// SIMATIC S7-200 project (STEP 7-Micro/WIN), CPU 226 REL 01.00

SYMBOL_TABLE SYM1
就联开关_就地甲I00      I0.0
就联开关_就地乙I01      I0.1
碎煤一开关_正转I02      I0.2
碎煤一开关_反转I03      I0.3
采样头开关_接通I04      I0.4
给料缩分机开关_接通I05    I0.5
提升螺旋机开关_接通I06    I0.6
联动信号甲I07         I0.7
联动信号乙I10         I1.0
采样甲限位I11         I1.1
采样乙限位I12         I1.2
分样机检测I13         I1.3
提升机热继I14         I1.4
螺旋机热继I15         I1.5
碎煤机一热继I16        I1.6
液压颚热继I17         I1.7
给料缩分机热继I20       I2.0
采样头甲热继I21        I2.1
采样头乙热继I22        I2.2
碎煤机二热继I23        I2.3
二级螺旋热继I24        I2.4
分样盘热继I25         I2.5
碎煤机一过流I26        I2.6
启动输入I27          I2.7
碎煤二开关_正转I30      I3.0
碎煤二开关_反转I31      I3.1
分样按钮_接通I32       I3.2
碎煤机二过流I33        I3.3
提升机_输出Q00        Q0.0
螺旋机_输出Q01        Q0.1
碎煤一正_输出QO2       Q0.2
碎煤一反_输出Q03       Q0.3
液压颚_输出Q04        Q0.4
给料机_输出Q05        Q0.5
采样甲_输出Q06        Q0.6
采样乙_输出Q07        Q0.7
缩分器_输出Q10        Q1.0
系统启动Q11          Q1.1
输煤带甲指示Q12        Q1.2
报警指示Q13          Q1.3
输煤带乙指示Q14        Q1.4
碎煤二正_输出Q16       Q1.6
碎煤二反_输出Q17       Q1.7
二级螺旋正_输出Q20      Q2.0
二级螺旋反_输出Q21      Q2.1
分样机_输出Q22        Q2.2
END_SYMBOL_TABLE

ORGANIZATION_BLOCK MAIN:OB1
TITLE=系统部署在洛河某燃煤处理车间。
// 采样过程从煤炭提升开始，提升机将煤炭送至高处，但只有在提升机热继未动作时才会启动，以保护设备。提升机在系统投运时，根据提升螺旋机开关_接通的状态启动，并通过运行指示显示其工作状态。随后，螺旋机在系统投运一段时间后（由计时触发），根据提升螺旋机开关_接通的状态并确保螺旋机热继正常，将煤炭输送至破碎区。螺旋机的运行状态通过显示实时反馈给操作员，确保输送过程可监控。
// 煤炭进入破碎环节，碎煤一正和碎煤二正依次破碎大块煤炭。若碎煤机一过流检测到堵塞，系统自动切换至碎煤一反反转排除故障，反转仅在过流或手动触发时发生，确保系统连续运行。碎煤一正的正转状态通过显示反馈，方便操作员确认破碎进程。破碎过程中，液压颚在碎煤一正运行时周期性动作，控制煤炭流量，其运行时间由液压间隔时间和击时间精确调节，避免设备过载。破碎后的煤炭通过给料机调节流量，进入采样区。
// 采样环节由采样甲和采样乙执行，根据采样间隔时间周期性采集样品，避免采样频率过高。采样甲完成标志在采样甲限位触发时记录，标记采样头甲的任务结束。采集的样品经缩分器处理后，由二级螺旋正输送，最终通过手动触发分样按钮_接通启动分样机。分样机在系统投运标志激活且采样完成后，根据分样按钮_接通的指令，将样品分配到不同容器中。分样机的运行状态通过显示提供给操作员，便于监控样品分配过程。每台设备的启动都依赖对应热继未动作，确保安全运行。若发生故障，如碎煤机一热继或碎煤机二过流，系统立即触发报警指示，报警状态持续显示，直到复位标志被触发以清除故障记录。复位标志在触发后清除故障记录，为系统恢复正常操作做准备，此时设备保持当前运行状态等待进一步操作。
// 
// 
BEGIN
Network 1 // 洛河入炉煤程序
// 段注释
// 
LD     SM5.0
STOP
Network 2
LD     SM0.1
LD     系统启动Q11:Q1.1
EU
OLD
R      M0.7, 1
R      M1.1, 1
R      M1.2, 1
R      M5.1, 1
R      M5.4, 1
Network 3
LDN    提升机热继I14:I1.4
AN     螺旋机热继I15:I1.5
AN     碎煤机一热继I16:I1.6
AN     液压颚热继I17:I1.7
AN     给料缩分机热继I20:I2.0
AN     采样头甲热继I21:I2.1
AN     采样头乙热继I22:I2.2
AN     碎煤机二热继I23:I2.3
AN     二级螺旋热继I24:I2.4
AN     分样盘热继I25:I2.5
=      M0.1
Network 4
LD     启动输入I27:I2.7
A      M0.1
AN     M5.0
TON    T101, +2
Network 5
LD     T101
=      系统启动Q11:Q1.1
Network 6 // 显待机
// 
// 
LD     系统启动Q11:Q1.1
AN     M2.0
BMB    VB420, VB40, 20
Network 7 // 显示停止
// 
// 
LDN    系统启动Q11:Q1.1
BMB    VB520, VB40, 20
Network 8 // 系统投运
// 
// 
LD     就联开关_就地甲I00:I0.0
O      就联开关_就地乙I01:I0.1
LDN    就联开关_就地甲I00:I0.0
AN     就联开关_就地乙I01:I0.1
LD     联动信号甲I07:I0.7
O      联动信号乙I10:I1.0
ALD
OLD
O      M2.0
A      系统启动Q11:Q1.1
AN     M1.4
=      M2.0
BMB    VB400, VB40, 10
TON    T127, +10
TON    T128, +20
TON    T129, +50
EU
R      M20.2, 1
R      M20.3, 1
Network 9 // 显示甲侧
// 
// 
LD     就联开关_就地甲I00:I0.0
BMB    VB740, VB260, 10
Network 10 // 显示乙侧
// 
// 
LD     就联开关_就地乙I01:I0.1
BMB    VB760, VB260, 10
Network 11 // 显示联动
// 
// 
LDN    就联开关_就地甲I00:I0.0
AN     就联开关_就地乙I01:I0.1
BMB    VB780, VB260, 10
Network 12 // 分计时器
// 
// 
LD     M2.0
AN     T115
TON    T115, +600
MOVW   T115, VW340
/I     +10, VW340
Network 13 // 一小时定时器
// 
// 
LD     T115
LD     C1
O      SM0.1
CTU    C1, +60
Network 14
LD     M2.0
MOVW   C1, VW342
Network 15
LD     M2.0
EU
MOVW   VW344, VW344
MOVW   +0, VW312
MOVW   +0, VW314
Network 16 // 累计运行时间记录
// 
// 
LD     C1
EU
INCW   VW344
INCW   VW346
Network 17 // 设置停机延时时间
// 
// 
LD     SM0.0
MOVW   VW396, AC0
MUL    +10, AC0
MOVW   AC0, VW398
Network 18 // 停运指令后启动30秒延时
// 
// 
LD     系统启动Q11:Q1.1
A      M2.0
AN     就联开关_就地甲I00:I0.0
AN     就联开关_就地乙I01:I0.1
AN     联动信号甲I07:I0.7
AN     联动信号乙I10:I1.0
TON    T113, VW398
Network 19 // M1.4去停机,T105为反排结束;如果碎煤机不在"正转"位置,就不执行反排动作而直接停机.
// 
// 
LD     T113
LDN    碎煤一开关_正转I02:I0.2
O      T105
ALD
LDN    碎煤二开关_正转I30:I3.0
O      T123
ALD
EU
=      M1.4
Network 20 // 甲启动状态，
// 
// 
LD     就联开关_就地甲I00:I0.0
=      M20.0
Network 21 // 乙启动状态，送远方Q2。5
// 
// 
LD     就联开关_就地乙I01:I0.1
=      M20.1
Network 22 // 甲侧初始状态
// 
// 
LDN    就联开关_就地甲I00:I0.0
AN     就联开关_就地乙I01:I0.1
A      联动信号甲I07:I0.7
A      M2.0
EU
AN     M20.3
S      M20.2, 1
R      M20.3, 1
Network 23 // 乙侧初始状态
// 
// 
LDN    就联开关_就地甲I00:I0.0
AN     就联开关_就地乙I01:I0.1
A      联动信号乙I10:I1.0
A      M2.0
EU
AN     M20.2
S      M20.3, 1
R      M20.2, 1
Network 24 // 双皮带同时运行情况，从双皮带变为单皮带情况。
// 
// 
LDN    就联开关_就地甲I00:I0.0
AN     就联开关_就地乙I01:I0.1
LPS
A      联动信号甲I07:I0.7
A      联动信号乙I10:I1.0
LPS
AN     M20.2
TON    T131, +18000
LRD
AN     M20.3
TON    T132, +18000
LRD
A      T131
S      M20.2, 1
R      M20.3, 1
LPP
A      T132
S      M20.3, 1
R      M20.2, 1
LPP
LPS
A      联动信号甲I07:I0.7
ED
S      M20.3, 1
R      M20.2, 1
LPP
A      联动信号乙I10:I1.0
ED
S      M20.2, 1
R      M20.3, 1
Network 25 // 二级螺旋
// 
// 
LD     M20.1
O      M20.3
A      M2.0
A      提升螺旋机开关_接通I06:I0.6
AN     二级螺旋热继I24:I2.4
AN     二级螺旋正_输出Q20:Q2.0
=      二级螺旋反_输出Q21:Q2.1
Network 26 // 二级螺旋正转指示
// 
// 
LD     二级螺旋正_输出Q20:Q2.0
LPS
A      SM0.6
LPS
AW<=   VW392, +0
MOVW   +100, VW392
LPP
DECW   VW392
LPP
NOT
MOVW   +0, VW392
Network 27 // 二级螺旋反转指示
// 
// 
LD     二级螺旋反_输出Q21:Q2.1
LPS
A      SM0.6
LPS
AW<=   VW394, +0
MOVW   +100, VW394
LPP
DECW   VW394
LPP
NOT
MOVW   +0, VW394
Network 28
LD     二级螺旋正_输出Q20:Q2.0
BMB    VB440, VB60, 20
Network 29
LD     二级螺旋反_输出Q21:Q2.1
BMB    VB460, VB60, 20
Network 30
LDN    二级螺旋正_输出Q20:Q2.0
AN     二级螺旋反_输出Q21:Q2.1
BMB    VB480, VB60, 20
Network 31 // 提升机启动.
// 
// 
LD     M2.0
A      提升螺旋机开关_接通I06:I0.6
AN     提升机热继I14:I1.4
LPS
=      提升机_输出Q00:Q0.0
A      SM0.6
LPS
AW<=   VW390, +0
MOVW   +100, VW390
LPP
DECW   VW390
LPP
NOT
MOVW   +100, VW390
Network 32 // 提升机运行
// 
// 
LD     提升机_输出Q00:Q0.0
BMB    VB500, VB80, 20
Network 33 // 提升机停机
// 
// 
LDN    提升机_输出Q00:Q0.0
AN     提升机热继I14:I1.4
BMB    VB520, VB80, 20
Network 34 // 提升机故障
// 
// 
LD     提升机热继I14:I1.4
BMB    VB540, VB80, 20
Network 35 // 螺旋机一启动.
// 
// 
LD     T127
AN     螺旋机热继I15:I1.5
A      提升螺旋机开关_接通I06:I0.6
=      螺旋机_输出Q01:Q0.1
Network 36 // 螺旋一运行
// 
// 
LD     螺旋机_输出Q01:Q0.1
BMB    VB500, VB100, 20
Network 37 // 螺旋一停机
// 
// 
LDN    螺旋机_输出Q01:Q0.1
AN     螺旋机热继I15:I1.5
BMB    VB520, VB100, 20
Network 38 // 螺旋一故障
// 
// 
LD     螺旋机热继I15:I1.5
BMB    VB540, VB100, 20
Network 39 // 碎煤机
// 
// 
LD     T128
A      碎煤一开关_正转I02:I0.2
AN     碎煤机一热继I16:I1.6
AN     M0.5
TON    T102, +20
A      T102
LPS
=      碎煤一正_输出QO2:Q0.2
A      SM0.6
LPS
AW<=   VW378, +0
MOVW   +100, VW378
LPP
DECW   VW378
LPP
NOT
MOVW   +0, VW378
Network 40 // 碎煤机过流防扰
// 
// 
LD     M2.0
A      碎煤机一过流I26:I2.6
A      碎煤一正_输出QO2:Q0.2
TON    T103, +10
Network 41 // 过流状态保持
// 
// 
LD     T103
O      M0.5
A      M2.0
AN     T105
O      T113
=      M0.5
TON    T104, +20
Network 42 // 手动反转时加延时
// 
// 
LD     碎煤一开关_反转I03:I0.3
A      M2.0
TON    T116, +20
Network 43 // 设置一级反排时间
// 
// 
LD     SM0.0
MOVW   VW372, AC0
MUL    +10, AC0
MOVW   AC0, VW374
Network 44 // 碎煤机反
// 
// 
LD     T104
O      T116
AN     碎煤机一热继I16:I1.6
AN     T106
=      碎煤一反_输出Q03:Q0.3
A      碎煤一开关_正转I02:I0.2
TON    T105, VW374
MOVW   T106, VW376
/I     +10, VW376
Network 45 // 反排期间过流
// 
// 
LD     碎煤一反_输出Q03:Q0.3
A      碎煤机一过流I26:I2.6
TON    T106, +20
Network 46 // 碎煤机报警
// 
// 
LD     T106
S      M0.7, 1
Network 47 // 碎煤正转显示
// 
// 
LD     碎煤一正_输出QO2:Q0.2
AN     碎煤机一过流I26:I2.6
BMB    VB560, VB120, 20
Network 48 // 碎煤反转显示
// 
// 
LD     碎煤一反_输出Q03:Q0.3
AN     碎煤机一过流I26:I2.6
BMB    VB580, VB120, 20
Network 49 // 碎煤停机显示
// 
// 
LDN    碎煤一正_输出QO2:Q0.2
AN     碎煤一反_输出Q03:Q0.3
AN     M0.7
AN     碎煤机一热继I16:I1.6
BMB    VB600, VB120, 20
Network 50 // 碎煤故障显示
// 
// 
LD     M0.7
O      碎煤机一热继I16:I1.6
BMB    VB620, VB120, 20
Network 51 // 碎煤过流显示
// 
// 
LD     碎煤一正_输出QO2:Q0.2
O      碎煤一反_输出Q03:Q0.3
A      碎煤机一过流I26:I2.6
BMB    VB640, VB120, 20
Network 52 // 设置液压间隔时间
// 
// 
LD     SM0.0
MOVW   VW358, AC0
MUL    +10, AC0
MOVW   AC0, VW360
Network 53 // 液压颚
// 
// 
LD     碎煤一正_输出QO2:Q0.2
AN     液压颚_输出Q04:Q0.4
TON    T126, VW360
MOVW   T126, VW362
/I     +10, VW362
Network 54 // 设置采液压颚击时间
// 
// 
LD     SM0.0
MOVW   VW364, AC0
MUL    +10, AC0
MOVW   AC0, VW366
Network 55 // 液压颚
// 
// 
LD     T126
O      液压颚_输出Q04:Q0.4
LD     M2.7
A      M3.2
OLD
A      M2.0
AN     T109
AN     液压颚热继I17:I1.7
LPS
=      液压颚_输出Q04:Q0.4
TON    T109, VW366
INCW   VW368
AW>    VW368, +100
MOVW   +100, VW368
LPP
NOT
MOVW   +0, VW368
Network 56 // 液压颚运行指示
// 
// 
LD     液压颚_输出Q04:Q0.4
BMB    VB660, VB140, 20
Network 57 // 液压颚停机指示
// 
// 
LDN    液压颚_输出Q04:Q0.4
AN     液压颚热继I17:I1.7
BMB    VB680, VB140, 20
Network 58 // 液压颚故障指示
// 
// 
LD     液压颚热继I17:I1.7
BMB    VB540, VB140, 20
Network 59 // 给料机
// 
// 
LD     T129
AN     给料缩分机热继I20:I2.0
A      给料缩分机开关_接通I05:I0.5
LPS
=      给料机_输出Q05:Q0.5
A      SM0.6
LPS
AW<=   VW370, +0
MOVW   +100, VW370
LPP
DECW   VW370
LPP
NOT
MOVW   +0, VW370
Network 60 // 给料机运行指示
// 
// 
LD     给料机_输出Q05:Q0.5
BMB    VB500, VB160, 20
Network 61 // 给料机停机指示
// 
// 
LDN    给料机_输出Q05:Q0.5
AN     给料缩分机热继I20:I2.0
BMB    VB520, VB160, 20
Network 62 // 给料机故障指示
// 
// 
LD     给料缩分机热继I20:I2.0
BMB    VB540, VB160, 20
Network 63 // 二级碎煤机
// 
// 
LD     M2.0
A      碎煤二开关_正转I30:I3.0
AN     碎煤机二热继I23:I2.3
AN     M0.2
TON    T120, +20
A      T120
LPS
=      碎煤二正_输出Q16:Q1.6
A      SM0.6
LPS
AW<=   VW386, +0
MOVW   +100, VW386
LPP
DECW   VW386
LPP
NOT
MOVW   +0, VW386
Network 64 // 二级碎煤机过流防扰
// 
// 
LD     M2.0
A      碎煤机二过流I33:I3.3
A      碎煤二正_输出Q16:Q1.6
TON    T121, +10
Network 65 // 过流状态保持
// 
// 
LD     T121
O      M0.2
A      M2.0
AN     T123
O      T113
=      M0.2
TON    T122, +20
Network 66 // 手动反转时加延时
// 
// 
LD     碎煤二开关_反转I31:I3.1
A      M2.0
TON    T124, +20
Network 67 // 设置二级反排时间
// 
// 
LD     SM0.0
MOVW   VW380, AC0
MUL    +10, AC0
MOVW   AC0, VW382
Network 68 // 二级碎煤机反
// 
// 
LD     T122
O      T124
AN     碎煤机二热继I23:I2.3
AN     T125
=      碎煤二反_输出Q17:Q1.7
A      碎煤二开关_正转I30:I3.0
TON    T123, VW382
MOVW   T123, VW384
/I     +10, VW384
Network 69 // 反排期间过流
// 
// 
LD     碎煤二反_输出Q17:Q1.7
A      碎煤机二过流I33:I3.3
TON    T125, +20
Network 70 // 二级碎煤机报警
// 
// 
LD     T125
S      M0.3, 1
Network 71 // 二级碎煤正转显示
// 
// 
LD     碎煤二正_输出Q16:Q1.6
AN     碎煤机二过流I33:I3.3
BMB    VB560, VB180, 20
Network 72 // 二级碎煤反转显示
// 
// 
LD     碎煤二反_输出Q17:Q1.7
AN     碎煤机二过流I33:I3.3
BMB    VB580, VB180, 20
Network 73 // 二级碎煤停机显示
// 
// 
LDN    碎煤二正_输出Q16:Q1.6
AN     碎煤二反_输出Q17:Q1.7
AN     M0.3
AN     碎煤机二热继I23:I2.3
BMB    VB600, VB180, 20
Network 74 // 二级碎煤故障显示
// 
// 
LD     M0.3
O      碎煤机二热继I23:I2.3
BMB    VB620, VB180, 20
Network 75 // 二级碎煤过流显示
// 
// 
LD     碎煤二正_输出Q16:Q1.6
O      碎煤二反_输出Q17:Q1.7
A      碎煤机二过流I33:I3.3
BMB    VB640, VB180, 20
Network 76 // 缩分器
// 
// 
LD     T128
A      给料缩分机开关_接通I05:I0.5
AN     给料缩分机热继I20:I2.0
LPS
=      缩分器_输出Q10:Q1.0
A      SM0.6
LPS
AW<=   VW388, +0
MOVW   +100, VW388
LPP
DECW   VW388
LPP
NOT
MOVW   +0, VW388
Network 77 // 设置采样间隔时间
// 
// 
LD     SM0.0
MOVW   VW350, AC0
MUL    +10, AC0
MOVW   AC0, VW352
Network 78 // 采样头
// 
// 
LD     M2.0
A      采样头开关_接通I04:I0.4
AN     T108
AN     M2.5
AN     M2.6
TON    T107, VW352
MOVW   T107, AC0
MUL    +100, AC0
DTR    AC0, AC0
XORD   AC1, AC1
MOVW   VW352, AC1
DTR    AC1, AC1
/R     AC1, AC0
TRUNC  AC0, VD354
NOT
MOVD   +0, VD354
Network 79 // 采样甲
// 
// 
LD     M20.0
O      M20.2
A      T107
LD     M2.7
A      M3.0
O      采样甲_输出Q06:Q0.6
OLD
AN     T108
AW<>   VW352, +0
AN     M2.5
=      采样甲_输出Q06:Q0.6
Network 80 // 采样乙
// 
// 
LD     M20.1
O      M20.3
A      T107
LD     M2.7
A      M3.1
O      采样乙_输出Q07:Q0.7
OLD
AN     T108
AW<>   VW352, +0
AN     M2.6
=      采样乙_输出Q07:Q0.7
Network 81 // 采样头定时保护
// 
// 
LD     采样甲_输出Q06:Q0.6
O      采样乙_输出Q07:Q0.7
TON    T108, +30
Network 82
LD     T108
LPS
A      采样甲_输出Q06:Q0.6
S      M1.1, 1
LPP
A      采样乙_输出Q07:Q0.7
S      M1.2, 1
Network 83 // 采样甲限位
// 
// 
LD     采样甲限位I11:I1.1
EU
=      M2.5
Network 84 // 采样乙限位
// 
// 
LD     采样乙限位I12:I1.2
EU
=      M2.6
Network 85 // 甲采样次数记录
// 
// 
LD     采样甲_输出Q06:Q0.6
EU
INCD   VD304
INCW   VW312
Network 86 // 乙采样次数记录
// 
// 
LD     采样乙_输出Q07:Q0.7
EU
INCD   VD308
INCW   VW314
Network 87 // 采样甲运行
// 
// 
LD     采样甲_输出Q06:Q0.6
BMB    VB700, VB220, 10
Network 88 // 采样甲停机
// 
// 
LDN    采样甲_输出Q06:Q0.6
AN     M1.1
AN     采样头甲热继I21:I2.1
BMB    VB720, VB220, 20
Network 89 // 采样甲故障
// 
// 
LD     M1.1
O      采样头甲热继I21:I2.1
BMB    VB540, VB220, 20
Network 90 // 采样乙运行
// 
// 
LD     采样乙_输出Q07:Q0.7
BMB    VB700, VB240, 20
Network 91 // 采样乙停机
// 
// 
LDN    采样乙_输出Q07:Q0.7
AN     M1.2
AN     采样头乙热继I22:I2.2
BMB    VB720, VB240, 20
Network 92 // 采样乙故障
// 
// 
LD     M1.2
O      采样头乙热继I22:I2.2
BMB    VB540, VB240, 20
Network 93 // 分样机
// 
// 
LD     M2.0
A      分样按钮_接通I32:I3.2
O      分样机_输出Q22:Q2.2
AN     M5.5
AN     分样盘热继I25:I2.5
A      系统启动Q11:Q1.1
LPS
=      分样机_输出Q22:Q2.2
TON    T130, +10
MOVW   +100, VW790
NOT
MOVW   +0, VW790
LPP
EU
INCW   VW792
AW>=   VW792, +7
MOVW   +1, VW792
Network 94
LD     T130
A      分样机检测I13:I1.3
=      M5.5
Network 95 // 分样机输出显示
// 
// 
LD     分样机_输出Q22:Q2.2
BMB    VB500, VB200, 20
Network 96 // 分样机停机显示
// 
// 
LDN    分样机_输出Q22:Q2.2
AN     分样盘热继I25:I2.5
BMB    VB520, VB200, 20
Network 97 // 分样机故障显示
// 
// 
LD     分样盘热继I25:I2.5
BMB    VB540, VB200, 20
Network 98 // 皮带甲运行指示
// 
// 
LD     联动信号甲I07:I0.7
LPS
=      输煤带甲指示Q12:Q1.2
A      SM0.6
CALL   SBR_0:SBR0
LPP
NOT
MOVW   +0, VW300
Network 99 // 皮带乙运行指示
// 
// 
LD     联动信号乙I10:I1.0
LPS
=      输煤带乙指示Q14:Q1.4
A      SM0.6
CALL   SBR_1:SBR1
LPP
NOT
MOVW   +0, VW302
Network 100 // 故障报警，利用"确认按钮M5.1"来关断报警声
// 
// 
LD     M0.7
O      M0.3
O      M1.1
O      M1.2
O      提升机热继I14:I1.4
O      螺旋机热继I15:I1.5
O      碎煤机一热继I16:I1.6
O      液压颚热继I17:I1.7
O      给料缩分机热继I20:I2.0
O      采样头甲热继I21:I2.1
O      采样头乙热继I22:I2.2
O      二级螺旋热继I24:I2.4
O      碎煤机二热继I23:I2.3
O      分样盘热继I25:I2.5
O      M5.4
LPS
AN     M5.1
AN     M2.1
=      报警指示Q13:Q1.3
TON    T111, +5
MOVW   +100, VW348
NOT
MOVW   +0, VW348
LPP
=      M5.0
Network 101
LD     T111
O      M2.1
AN     T112
TON    T112, +5
=      M2.1
Network 102 // 报警复位
// 
// 
LD     M5.2
LPS
A      M0.7
R      M0.7, 1
LRD
A      M0.3
R      M0.3, 1
LRD
A      M1.1
R      M1.1, 1
LRD
A      M1.2
R      M1.2, 1
LRD
R      M5.1, 1
LPP
A      M5.4
R      M5.4, 1
Network 103 // 读取系统日期时钟送入TP显示，VB10~VB15为16进制，VB20~VB31为ASCII码。
// 
// 
LD     SM0.0
TODR   VB10
HTA    VB10, VB20, 2
HTA    VB11, VB22, 2
HTA    VB12, VB24, 2
HTA    VB13, VB26, 2
HTA    VB14, VB28, 2
HTA    VB15, VB30, 2
Network 104
LD     M3.5
TODW   VB0
END_ORGANIZATION_BLOCK

SUBROUTINE_BLOCK SBR_0:SBR0
TITLE= 
// 子程序注释
// 按 F1 获得帮助及举例程序
//  
BEGIN
Network 1 // 网络题目 (单行)
//  
// 网络注释
//  
// 
LDN    M1.5
+I     +10, VW300
AW>=   VW300, +100
S      M1.5, 1
R      M1.6, 1
Network 2
LDN    M1.6
-I     +10, VW300
AW<=   VW300, +10
S      M1.6, 1
R      M1.5, 1
END_SUBROUTINE_BLOCK

SUBROUTINE_BLOCK SBR_1:SBR1
TITLE= 
// 子程序注释
// 按 F1 获得帮助及举例程序
//  
BEGIN
Network 1 // 网络题目 (单行)
//  
// 网络注释
//  
// 
LDN    M1.3
+I     +10, VW302
AW>=   VW302, +100
S      M1.3, 1
R      M1.7, 1
Network 2
LDN    M1.7
-I     +10, VW302
AW<=   VW302, +10
S      M1.7, 1
R      M1.3, 1
Network 3 // 网络题目 (单行)
//  
// 网络注释
//  
// 
END_SUBROUTINE_BLOCK

DATA_BLOCK_TAB USER1
BEGIN
VW330    30
VB400    'Start'
VB420    'StandBy'
VB440    'PositionNo.1'
VB460    'PositionNo.2'
VB480    'In the middle'
VB500    'Run!'
VB520    'Stop!'
VB540    'trouble!'
VB560    'Turning!'
VB580    'Reverse!'
VB600    'Stop!'
VB620    'Trouble'
VB660    'Push!'
VB680    'Stop!'
VB700    'Sample'
VB720    'Stop!'
VB740    'LocalNo1'
VB760    'LocalNo2'
VB780    'Interlock'
END_DATA_BLOCK_TAB
